// A class with helper methods when working with files.
{attribute 'no_explicit_call' := 'Body contains no logic, calling methods only allowed.'}
PROGRAM Utilities

VAR
	_directory	: FB_DirectoryUtilities;
	_file		: FB_FileUtilities;
	_path		: FB_PathUtilities;
END_VAR

PROPERTY Directory : I_Directory
GET
Directory := _directory;
END_GET
END_PROPERTY

PROPERTY File : I_File
GET
File := _file;
END_GET
END_PROPERTY

PROPERTY Path : I_Path
GET
Path := _path;
END_GET
END_PROPERTY

END_PROGRAM

(* stored: Version 1.1.0.1, ProductVersion 3.1.4024.15
   POU Utilities: Id {6ee3af3c-bb5a-0bbf-0e0a-dc339ace1c34}, SpecialFunc None
   Property Directory: Id {b5c2a1fb-dcb0-04a9-13ed-747fa10f323b}
   Get Get: Id {e8866c8d-9c03-07f7-0393-6d6ca370781a}
   Property File: Id {b8d87f58-37b0-00fd-299e-7b66a103005d}
   Get Get: Id {65d0bf53-4594-01a5-3f01-a29ab15e096d}
   Property Path: Id {caf0782a-5710-0ee3-3205-abcccb7a7715}
   Get Get: Id {99e43f93-ab59-0d38-3eef-4e36c7050dcb} *)
